# EPICS substitutions: iocLinkam/asynRecord.substitutions
file "$(ASYN)/db/asynRecord.db"
{
pattern
{P        R         PORT    ADDR    OMAX  IMAX}
{dp_linkam_xrd47:     asyn_1   serial1    0     256  256}
#{dp_linkam_xrd47:     asyn_2   serial2    0     256  256}
#{dp_linkam_xrd47:     asyn_3   serial3    0     256  256}
#{dp_linkam_xrd47:     asyn_4   serial4    0     256  256}
}
